INTERFACE I_CommandStepParser

METHOD AssemblyEndParse : BOOL

VAR_INPUT
    Step          : ST_CSV_Step;
    StepDetailOut : REFERENCE TO ST_AssemblyEnd;
END_VAR
END_METHOD

METHOD AssemblyStartParse : BOOL
VAR_INPUT
    Step    : ST_CSV_Step;
    StepOut : REFERENCE TO ST_AssemblyStart;
END_VAR
END_METHOD

METHOD BoardInfoParse : BOOL
VAR_INPUT
    Step    : ST_CSV_Step;
    StepOut : REFERENCE TO ST_BoardInfo;
END_VAR
END_METHOD

METHOD BoardParse : BOOL
VAR_INPUT
    Step    : ST_CSV_Step;
    StepOut : REFERENCE TO ST_Board;
END_VAR
END_METHOD

METHOD NailPlateParse : BOOL
VAR_INPUT
    Step    : ST_CSV_Step;
    StepOut : REFERENCE TO ST_BoardInfo;
END_VAR
END_METHOD

METHOD TrussInfoParse : BOOL
VAR_INPUT
    Step    : ST_CSV_Step;
    StepOut : REFERENCE TO ST_TrussInfo;
END_VAR
END_METHOD

END_INTERFACE

(* stored: Version 1.1.0.1
   Itf I_CommandStepParser: Id {780b93d5-ee76-4b0a-a5a7-3a041d38f4cf}
   Method AssemblyEndParse: Id {722dea96-eb4a-4273-b71d-372bbe543b92}
   Method AssemblyStartParse: Id {6e4cbf22-84c0-40b3-910b-b7bb7716ba2c}
   Method BoardInfoParse: Id {b618ac8d-dc30-4656-b711-a5e4382cef1f}
   Method BoardParse: Id {7dd8f931-da09-4fd9-85fb-aa51ac2ee8ff}
   Method NailPlateParse: Id {672f408d-2c55-4c86-8dc9-9798e4f146c8}
   Method TrussInfoParse: Id {c9b1a93c-4891-47f8-ad33-6f5cd37c5c4d} *)
